# EPICS autosave request: iocs/tpx3IOC/iocBoot/iocTimePix/profiles/tpx3/auto_settings.req
file "ADTimePix_settings.req",  P=$(P),  R=cam1:
file "NDStdArrays_settings.req",  P=$(P),  R=image1:
file "commonPlugin_settings.req", P=$(P)
